// TIA Portal V15.1 export
// export: Created 2024-05-17T05:38:33.3837164Z, ExportSetting WithDefaults, DisplayName Totally Integrated Automation Portal, DisplayVersion V15.1 Update 5, DisplayName TIA Portal Openness, DisplayVersion V15.1 Update 5, DisplayName SINAMICS Startdrive Advanced, DisplayVersion V15.1, DisplayName G130, G150, S120, S150, SINAMICS MV, S210, DisplayVersion V15.1, DisplayName G110M, G120, G120C, G120D, G120P, DisplayVersion V15.1, DisplayName STEP 7 Professional, DisplayVersion V15.1 Update 5, DisplayName STEP 7 Safety, DisplayVersion V15.1, DisplayName WinCC Professional, DisplayVersion V15.1 Update 5, DisplayName SIMATIC Visualization Architect, DisplayVersion V15.1
FUNCTION_BLOCK "LProcEntalphie"   // FB1718, STL
TITLE = LProcEnthalpie
{ S7_Optimized_Access := 'FALSE' }
AUTHOR : VCC
FAMILY : ProcEq
VERSION : 0.1
// This function is made for the calculatin of the Ethalpie from the temperature 
// and humidity measurements.
// stored: AutoNumber false, UDAEnableTagReadback false
   VAR_INPUT
      PvHumidity { ExternalAccessible := 'False'; ExternalVisible := 'False'; ExternalWritable := 'False'} : Real;   // Analoge input value humidity
      PvTemperature { ExternalAccessible := 'False'; ExternalVisible := 'False'; ExternalWritable := 'False'} : Real;   // Analoge intup value temperature
   END_VAR
   VAR_OUTPUT
      PvEnthalpie { ExternalAccessible := 'False'; ExternalVisible := 'False'; ExternalWritable := 'False'} : Real;   // Enthalpy calculation
   END_VAR
   VAR DB_SPECIFIC
      PvX { ExternalAccessible := 'False'; ExternalVisible := 'False'; ExternalWritable := 'False'} : Real;   // Humidity absolute for the process value
      PvPs { ExternalAccessible := 'False'; ExternalVisible := 'False'; ExternalWritable := 'False'} : Real;   // Value for steam pressure for the humidity value
      PvNbXYpoints { ExternalAccessible := 'False'; ExternalVisible := 'False'; ExternalWritable := 'False'} : Int;   // Edit number of X-Y points used
      PvFraction { ExternalAccessible := 'False'; ExternalVisible := 'False'; ExternalWritable := 'False'} : Int;
      PvBias { ExternalAccessible := 'False'; ExternalVisible := 'False'; ExternalWritable := 'False'} : Real;
      xl { ExternalAccessible := 'False'; ExternalVisible := 'False'; ExternalWritable := 'False'} : Real;
      xh { ExternalAccessible := 'False'; ExternalVisible := 'False'; ExternalWritable := 'False'} : Real;
      yl { ExternalAccessible := 'False'; ExternalVisible := 'False'; ExternalWritable := 'False'} : Real;
      yh { ExternalAccessible := 'False'; ExternalVisible := 'False'; ExternalWritable := 'False'} : Real;
      PvPstemp1 { ExternalAccessible := 'False'; ExternalVisible := 'False'; ExternalWritable := 'False'} : Real;
      PvPsTemp2 { ExternalAccessible := 'False'; ExternalVisible := 'False'; ExternalWritable := 'False'} : Real;
      PvPsTemp3 { ExternalAccessible := 'False'; ExternalVisible := 'False'; ExternalWritable := 'False'} : Real;
      PvXTemp1 { ExternalAccessible := 'False'; ExternalVisible := 'False'; ExternalWritable := 'False'} : Real;
      PvxTemp2 { ExternalAccessible := 'False'; ExternalVisible := 'False'; ExternalWritable := 'False'} : Real;
      PvXTemp3 { ExternalAccessible := 'False'; ExternalVisible := 'False'; ExternalWritable := 'False'} : Real;
      PvEnthTemp1 { ExternalAccessible := 'False'; ExternalVisible := 'False'; ExternalWritable := 'False'} : Real;
      PvEnthTemp2 { ExternalAccessible := 'False'; ExternalVisible := 'False'; ExternalWritable := 'False'} : Real;
   END_VAR
BEGIN

NETWORK
TITLE = **** 4.4 - Machine status - Calculation **** Calculate position
// Calculate position
      L     -10.0;
      T     #xl;
      L     260.0;
      T     #yl;
      L     0.0;
      T     #xh;
      L     610.59;
      T     #yh;






NETWORK
TITLE = **** 4.4 - Machine status - Calculation **** Calculate position
// Calculate position
      A(;
      L     #PvTemperature;
      L     0.0;
      >R;
      );
      JCN   End1;
      L     #xh;
      T     #xl;
      L     #yh;
      T     #yl;
      L     6.0;
      T     #xh;
      L     934.59;
      T     #yh;

End1: NOP   0;





NETWORK
TITLE = **** 4.4 - Machine status - Calculation **** Calculate position
// Calculate position
      A(;
      L     #PvTemperature;
      L     6.0;
      >R;
      );
      JCN   End2;
      L     #xh;
      T     #xl;
      L     #yh;
      T     #yl;
      L     12.0;
      T     #xh;
      L     1402.5;
      T     #yh;

End2: NOP   0;




NETWORK
TITLE = **** 4.4 - Machine status - Calculation **** Calculate position
// Calculate position
      A(;
      L     #PvTemperature;
      L     12.0;
      >R;
      );
      JCN   End3;
      L     #xh;
      T     #xl;
      L     #yh;
      T     #yl;
      L     16.0;
      T     #xh;
      L     1817.2;
      T     #yh;

End3: NOP   0;





NETWORK
TITLE = **** 4.4 - Machine status - Calculation **** Calculate position
// Calculate position
      A(;
      L     #PvTemperature;
      L     16.0;
      >R;
      );
      JCN   End4;
      L     #xh;
      T     #xl;
      L     #yh;
      T     #yl;
      L     20.0;
      T     #xh;
      L     2337.1;
      T     #yh;

End4: NOP   0;





NETWORK
TITLE = **** 4.4 - Machine status - Calculation **** Calculate position
// Calculate position
      A(;
      L     #PvTemperature;
      L     20.0;
      >R;
      );
      JCN   End5;
      L     #xh;
      T     #xl;
      L     #yh;
      T     #yl;
      L     22.0;
      T     #xh;
      L     2643.8;
      T     #yh;

End5: NOP   0;




NETWORK
TITLE = **** 4.4 - Machine status - Calculation **** Calculate position
// Calculate position
      A(;
      L     #PvTemperature;
      L     22.0;
      >R;
      );
      JCN   End6;
      L     #xh;
      T     #xl;
      L     #yh;
      T     #yl;
      L     26.0;
      T     #xh;
      L     3361.0;
      T     #yh;

End6: NOP   0;





NETWORK
TITLE = **** 4.4 - Machine status - Calculation **** Calculate position
// Calculate position
      A(;
      L     #PvTemperature;
      L     26.0;
      >R;
      );
      JCN   End7;
      L     #xh;
      T     #xl;
      L     #yh;
      T     #yl;
      L     32.0;
      T     #xh;
      L     4754.3;
      T     #yh;

End7: NOP   0;





NETWORK
TITLE = **** 4.4 - Machine status - Calculation **** Calculate position
// Calculate position
      A(;
      L     #PvTemperature;
      L     32.0;
      >R;
      );
      JCN   End8;
      L     #xh;
      T     #xl;
      L     #yh;
      T     #yl;
      L     40.0;
      T     #xh;
      L     7375.4;
      T     #yh;

End8: NOP   0;




NETWORK
TITLE = **** 4.4 - Machine status - Calculation **** Process value Enthalpie
// Process value Enthalpie
      L     #xh;
      L     #xl;
      -R;
      ABS;
      L     0.0001;
      <R;
      JC    then;
      L     #yh;
      L     #yl;
      -R;
      T     #PvPstemp1;
      L     #xh;
      L     #xl;
      -R;
      T     #PvPsTemp2;
      L     #PvTemperature;
      L     #xl;
      -R;
      T     #PvPsTemp3;
      L     #PvPstemp1;
      L     #PvPsTemp2;
      /R;
      L     #PvPsTemp3;
      *R;
      L     #yl;
      +R;
      L     #PvBias;
      +R;
      T     #PvPs;
      JU    End;

then: L     #yh;
      L     #yl;
      +R;
      L     2.0;
      /R;
      L     #PvBias;
      +R;
      T     #PvPs;


End:  NOP   0;




NETWORK
TITLE = **** 4.4 - Machine status - Calculation **** Humidity absolut
// Humidity absolut
      L     0.622;
      L     #PvHumidity;
      *R;
      L     100.0;
      /R;
      L     #PvPs;
      *R;
      T     #PvXTemp1;
      L     #PvHumidity;
      L     100.0;
      /R;
      L     #PvPs;
      *R;
      T     #PvxTemp2;
      L     101356.9;
      L     #PvxTemp2;
      -R;
      T     #PvXTemp3;
      L     #PvXTemp1;
      L     #PvXTemp3;
      /R;
      T     #PvX;




NETWORK
TITLE = **** 4.4 - Machine status - Calculation **** Calculation of the process enthalpie value
// Calculation of the process enthalpie value
      L     2500.8;
      L     #PvX;
      *R;
      T     #PvEnthTemp1;
      L     1.927;
      L     #PvX;
      *R;
      L     #PvTemperature;
      *R;
      T     #PvEnthTemp2;
      L     1.006;
      L     #PvTemperature;
      *R;
      L     #PvEnthTemp1;
      +R;
      L     #PvEnthTemp2;
      +R;
      T     #PvEnthalpie;




END_FUNCTION_BLOCK
